// TIA Portal V21 export
FUNCTION_BLOCK "AiFb"   // FB108, LAD
{ S7_Optimized_Access := 'TRUE' }
// stored: AutoNumber false, MemoryReserve 100, SetENOAutomatically false
   VAR
      Ai01 { S7_SetPoint := 'True'} : "FB:Analog_Scaling";   // NfcoLineTemp(Ticr01)
      Ai02 { S7_SetPoint := 'True'} : "FB:Analog_Scaling";   // VfcoLineTemp(Ticr02)
      Ai03 { S7_SetPoint := 'True'} : "FB:Analog_Scaling";   // AiSpare01
      Ai04 { S7_SetPoint := 'True'} : "FB:Analog_Scaling";   // AiSpare02
      Ai05 { S7_SetPoint := 'True'} : "FB:Analog_Scaling";   // AiSpare03
      Ai06 { S7_SetPoint := 'True'} : "FB:Analog_Scaling";   // Pf01InLineTemp(Ticr06)
      Ai07 { S7_SetPoint := 'True'} : "FB:Analog_Scaling";   // Pf02InLineTemp(Ticr07)
      Ai08 { S7_SetPoint := 'True'} : "FB:Analog_Scaling";   // Pf02OutLineTemp(Ticr08)
      Ai09 { S7_SetPoint := 'True'} : "FB:Analog_Scaling";   // PtlDrainTemp(Ticr09)
      Ai10 { S7_SetPoint := 'True'} : "FB:Analog_Scaling";   // VesselTemp(Ticr10)
      Ai11 { S7_SetPoint := 'True'} : "FB:Analog_Scaling";   // VesselPressure(Picr01)
      Ai12 { S7_SetPoint := 'True'} : "FB:Analog_Scaling";   // VesselRclLine(Picr02)
      Ai13 { S7_SetPoint := 'True'} : "FB:Analog_Scaling";   // Pf01OutLinePressure(Picr03)
      Ai14 { S7_SetPoint := 'True'} : "FB:Analog_Scaling";   // Pf02OutLinePressure(Picr04)
      Ai15 { S7_SetPoint := 'True'} : "FB:Analog_Scaling";   // ProcessDrainConductivity
      Ai16 { S7_SetPoint := 'True'} : "FB:Analog_Scaling";   // AiSpare04
      Ai17 { S7_SetPoint := 'True'} : "FB:Analog_Scaling";   // AiSpare05
      Ai18 { S7_SetPoint := 'True'} : "FB:Analog_Scaling";   // AiSpare06
      Ai19 { S7_SetPoint := 'True'} : "FB:Analog_Scaling";   // AiSpare07
      Ai20 { S7_SetPoint := 'True'} : "FB:Analog_Scaling";   // AiSpare08
      Ai21 { S7_SetPoint := 'True'} : "FB:Analog_Scaling";   // AiSpare09
      Ai22 { S7_SetPoint := 'True'} : "FB:Analog_Scaling";   // AiSpare10
      Ai23 { S7_SetPoint := 'True'} : "FB:Analog_Scaling";   // AiSpare11
      Ai24 { S7_SetPoint := 'True'} : "FB:Analog_Scaling";   // AiSpare12
   END_VAR
BEGIN

REGION Network 1: #Ai01--- NfcoLineTemp
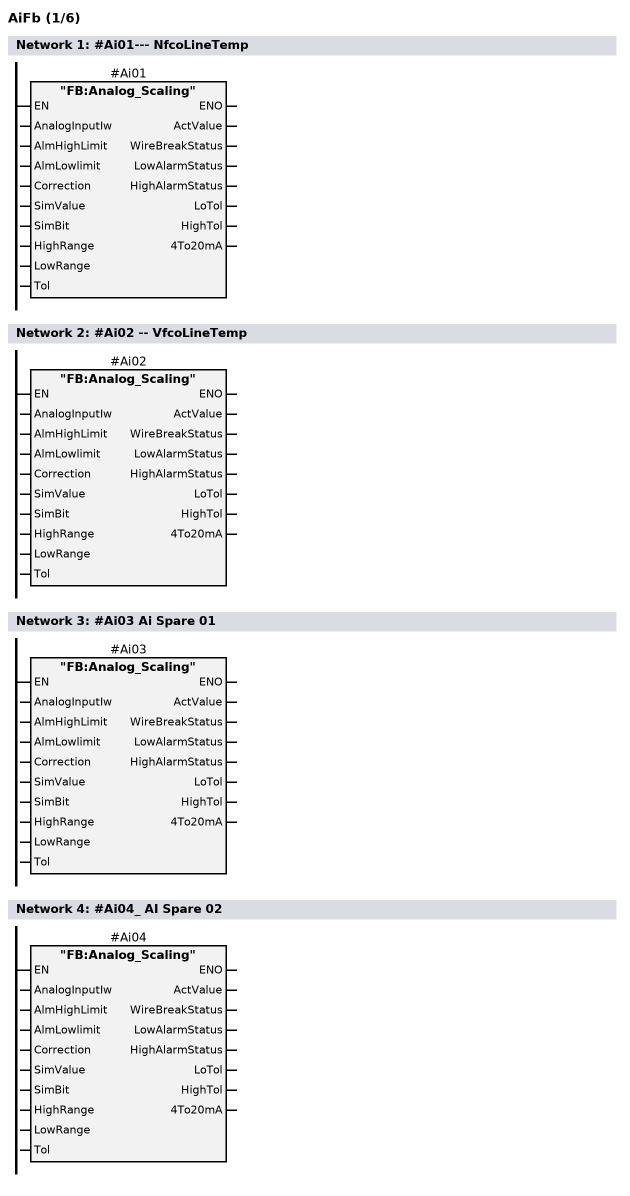
   RUNG wire#powerrail
      #Ai01(AnalogInputIw :=, AlmHighLimit :=, AlmLowlimit :=, Correction :=, SimValue :=, SimBit :=, HighRange :=, LowRange :=, Tol :=, ActValue =>, WireBreakStatus =>, LowAlarmStatus =>, HighAlarmStatus =>, LoTol =>, HighTol =>, "4To20mA" =>)
   END_RUNG
   // the same network as SCL:
   #Ai01();   // "FB:Analog_Scaling"
END_REGION

REGION Network 2: #Ai02 -- VfcoLineTemp
   RUNG wire#powerrail
      #Ai02(AnalogInputIw :=, AlmHighLimit :=, AlmLowlimit :=, Correction :=, SimValue :=, SimBit :=, HighRange :=, LowRange :=, Tol :=, ActValue =>, WireBreakStatus =>, LowAlarmStatus =>, HighAlarmStatus =>, LoTol =>, HighTol =>, "4To20mA" =>)
   END_RUNG
   // the same network as SCL:
   #Ai02();   // "FB:Analog_Scaling"
END_REGION

REGION Network 3: #Ai03 Ai Spare 01
   RUNG wire#powerrail
      #Ai03(AnalogInputIw :=, AlmHighLimit :=, AlmLowlimit :=, Correction :=, SimValue :=, SimBit :=, HighRange :=, LowRange :=, Tol :=, ActValue =>, WireBreakStatus =>, LowAlarmStatus =>, HighAlarmStatus =>, LoTol =>, HighTol =>, "4To20mA" =>)
   END_RUNG
   // the same network as SCL:
   #Ai03();   // "FB:Analog_Scaling"
END_REGION

REGION Network 4: #Ai04_ AI Spare 02
   RUNG wire#powerrail
      #Ai04(AnalogInputIw :=, AlmHighLimit :=, AlmLowlimit :=, Correction :=, SimValue :=, SimBit :=, HighRange :=, LowRange :=, Tol :=, ActValue =>, WireBreakStatus =>, LowAlarmStatus =>, HighAlarmStatus =>, LoTol =>, HighTol =>, "4To20mA" =>)
   END_RUNG
   // the same network as SCL:
   #Ai04();   // "FB:Analog_Scaling"
END_REGION

REGION Network 5: #Ai05--- #Ai04_ AI Spare 03
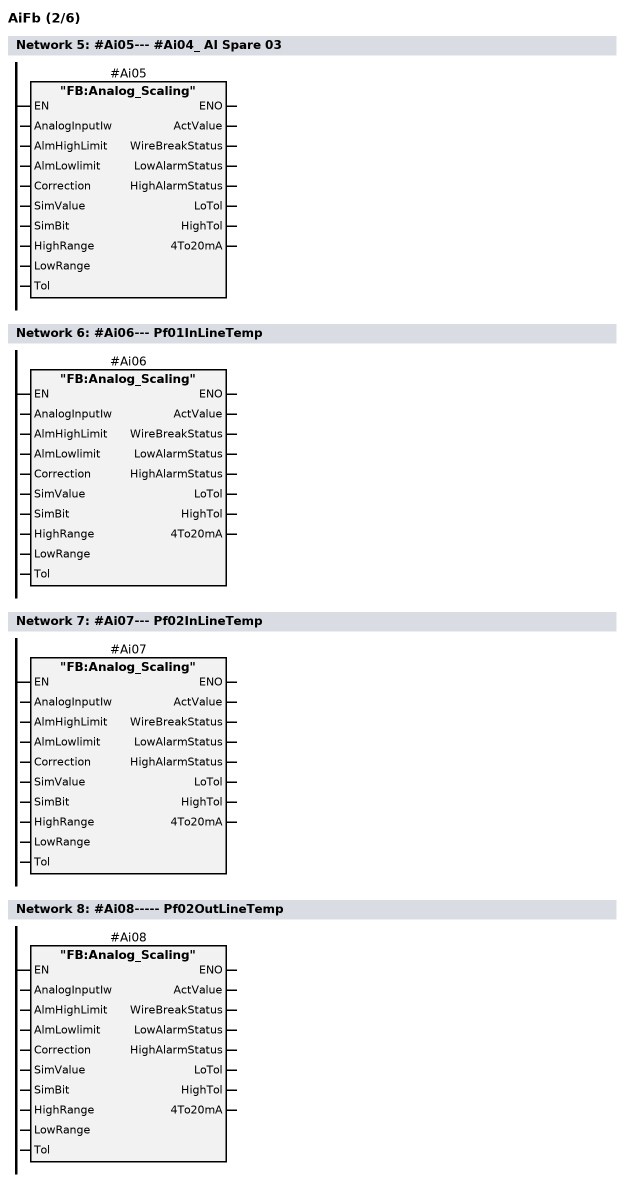
   RUNG wire#powerrail
      #Ai05(AnalogInputIw :=, AlmHighLimit :=, AlmLowlimit :=, Correction :=, SimValue :=, SimBit :=, HighRange :=, LowRange :=, Tol :=, ActValue =>, WireBreakStatus =>, LowAlarmStatus =>, HighAlarmStatus =>, LoTol =>, HighTol =>, "4To20mA" =>)
   END_RUNG
   // the same network as SCL:
   #Ai05();   // "FB:Analog_Scaling"
END_REGION

REGION Network 6: #Ai06--- Pf01InLineTemp
   RUNG wire#powerrail
      #Ai06(AnalogInputIw :=, AlmHighLimit :=, AlmLowlimit :=, Correction :=, SimValue :=, SimBit :=, HighRange :=, LowRange :=, Tol :=, ActValue =>, WireBreakStatus =>, LowAlarmStatus =>, HighAlarmStatus =>, LoTol =>, HighTol =>, "4To20mA" =>)
   END_RUNG
   // the same network as SCL:
   #Ai06();   // "FB:Analog_Scaling"
END_REGION

REGION Network 7: #Ai07--- Pf02InLineTemp
   RUNG wire#powerrail
      #Ai07(AnalogInputIw :=, AlmHighLimit :=, AlmLowlimit :=, Correction :=, SimValue :=, SimBit :=, HighRange :=, LowRange :=, Tol :=, ActValue =>, WireBreakStatus =>, LowAlarmStatus =>, HighAlarmStatus =>, LoTol =>, HighTol =>, "4To20mA" =>)
   END_RUNG
   // the same network as SCL:
   #Ai07();   // "FB:Analog_Scaling"
END_REGION

REGION Network 8: #Ai08----- Pf02OutLineTemp
   RUNG wire#powerrail
      #Ai08(AnalogInputIw :=, AlmHighLimit :=, AlmLowlimit :=, Correction :=, SimValue :=, SimBit :=, HighRange :=, LowRange :=, Tol :=, ActValue =>, WireBreakStatus =>, LowAlarmStatus =>, HighAlarmStatus =>, LoTol =>, HighTol =>, "4To20mA" =>)
   END_RUNG
   // the same network as SCL:
   #Ai08();   // "FB:Analog_Scaling"
END_REGION

REGION Network 9: #Ai09---- PtlDrainTemp
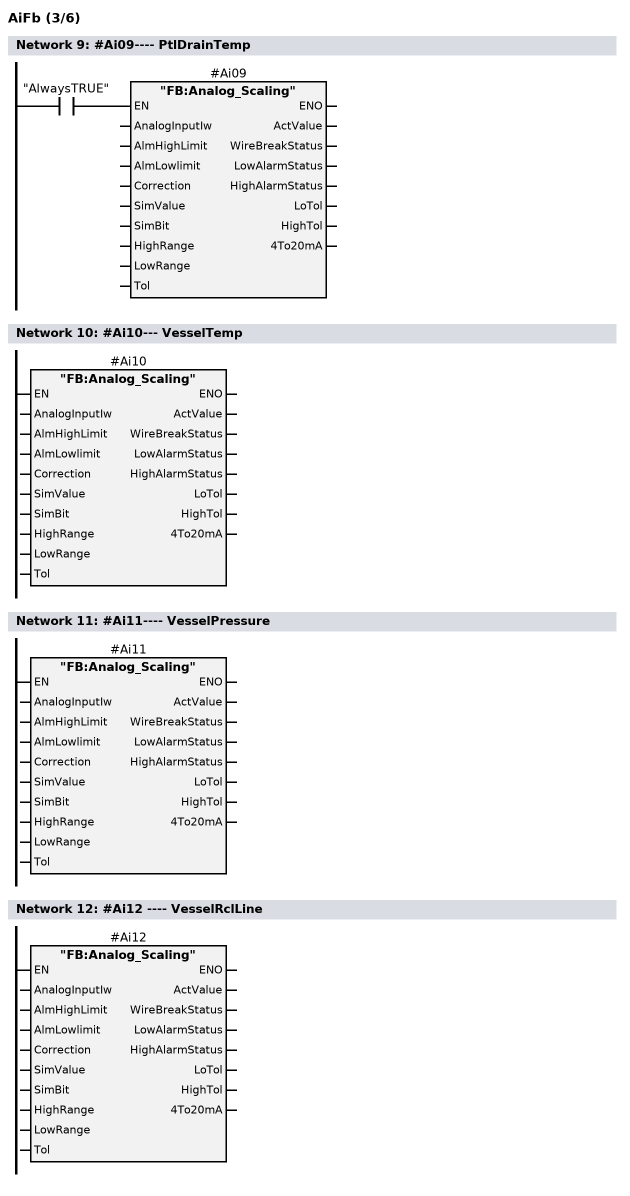
   RUNG wire#powerrail
      Contact( "AlwaysTRUE" )
      #Ai09(AnalogInputIw :=, AlmHighLimit :=, AlmLowlimit :=, Correction :=, SimValue :=, SimBit :=, HighRange :=, LowRange :=, Tol :=, ActValue =>, WireBreakStatus =>, LowAlarmStatus =>, HighAlarmStatus =>, LoTol =>, HighTol =>, "4To20mA" =>)
   END_RUNG
   // the same network as SCL:
   IF "AlwaysTRUE" THEN
       #Ai09();   // "FB:Analog_Scaling"
   END_IF;
END_REGION

REGION Network 10: #Ai10--- VesselTemp
   RUNG wire#powerrail
      #Ai10(AnalogInputIw :=, AlmHighLimit :=, AlmLowlimit :=, Correction :=, SimValue :=, SimBit :=, HighRange :=, LowRange :=, Tol :=, ActValue =>, WireBreakStatus =>, LowAlarmStatus =>, HighAlarmStatus =>, LoTol =>, HighTol =>, "4To20mA" =>)
   END_RUNG
   // the same network as SCL:
   #Ai10();   // "FB:Analog_Scaling"
END_REGION

REGION Network 11: #Ai11---- VesselPressure
   RUNG wire#powerrail
      #Ai11(AnalogInputIw :=, AlmHighLimit :=, AlmLowlimit :=, Correction :=, SimValue :=, SimBit :=, HighRange :=, LowRange :=, Tol :=, ActValue =>, WireBreakStatus =>, LowAlarmStatus =>, HighAlarmStatus =>, LoTol =>, HighTol =>, "4To20mA" =>)
   END_RUNG
   // the same network as SCL:
   #Ai11();   // "FB:Analog_Scaling"
END_REGION

REGION Network 12: #Ai12 ---- VesselRclLine
   RUNG wire#powerrail
      #Ai12(AnalogInputIw :=, AlmHighLimit :=, AlmLowlimit :=, Correction :=, SimValue :=, SimBit :=, HighRange :=, LowRange :=, Tol :=, ActValue =>, WireBreakStatus =>, LowAlarmStatus =>, HighAlarmStatus =>, LoTol =>, HighTol =>, "4To20mA" =>)
   END_RUNG
   // the same network as SCL:
   #Ai12();   // "FB:Analog_Scaling"
END_REGION

REGION Network 13: #Ai13--- Pf01OutLinePressure
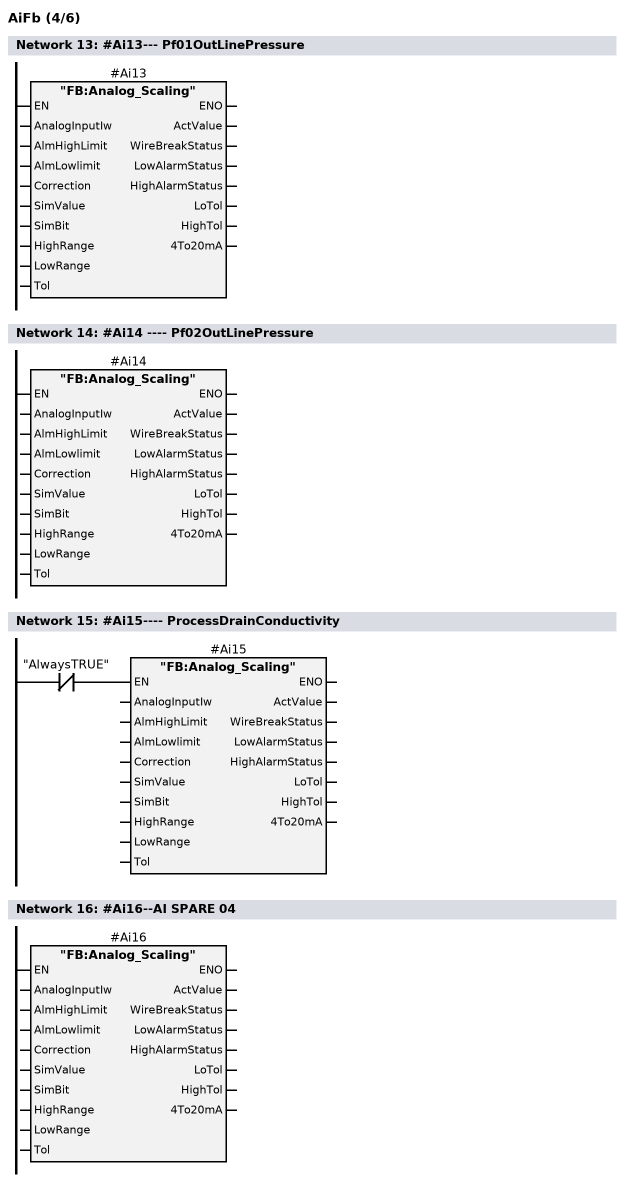
   RUNG wire#powerrail
      #Ai13(AnalogInputIw :=, AlmHighLimit :=, AlmLowlimit :=, Correction :=, SimValue :=, SimBit :=, HighRange :=, LowRange :=, Tol :=, ActValue =>, WireBreakStatus =>, LowAlarmStatus =>, HighAlarmStatus =>, LoTol =>, HighTol =>, "4To20mA" =>)
   END_RUNG
   // the same network as SCL:
   #Ai13();   // "FB:Analog_Scaling"
END_REGION

REGION Network 14: #Ai14 ---- Pf02OutLinePressure
   RUNG wire#powerrail
      #Ai14(AnalogInputIw :=, AlmHighLimit :=, AlmLowlimit :=, Correction :=, SimValue :=, SimBit :=, HighRange :=, LowRange :=, Tol :=, ActValue =>, WireBreakStatus =>, LowAlarmStatus =>, HighAlarmStatus =>, LoTol =>, HighTol =>, "4To20mA" =>)
   END_RUNG
   // the same network as SCL:
   #Ai14();   // "FB:Analog_Scaling"
END_REGION

REGION Network 15: #Ai15---- ProcessDrainConductivity
   RUNG wire#powerrail
      I_Contact( "AlwaysTRUE" )
      #Ai15(AnalogInputIw :=, AlmHighLimit :=, AlmLowlimit :=, Correction :=, SimValue :=, SimBit :=, HighRange :=, LowRange :=, Tol :=, ActValue =>, WireBreakStatus =>, LowAlarmStatus =>, HighAlarmStatus =>, LoTol =>, HighTol =>, "4To20mA" =>)
   END_RUNG
   // the same network as SCL:
   IF NOT "AlwaysTRUE" THEN
       #Ai15();   // "FB:Analog_Scaling"
   END_IF;
END_REGION

REGION Network 16: #Ai16--AI SPARE 04
   RUNG wire#powerrail
      #Ai16(AnalogInputIw :=, AlmHighLimit :=, AlmLowlimit :=, Correction :=, SimValue :=, SimBit :=, HighRange :=, LowRange :=, Tol :=, ActValue =>, WireBreakStatus =>, LowAlarmStatus =>, HighAlarmStatus =>, LoTol =>, HighTol =>, "4To20mA" =>)
   END_RUNG
   // the same network as SCL:
   #Ai16();   // "FB:Analog_Scaling"
END_REGION

REGION Network 17: #Ai17--AI SPARE 05
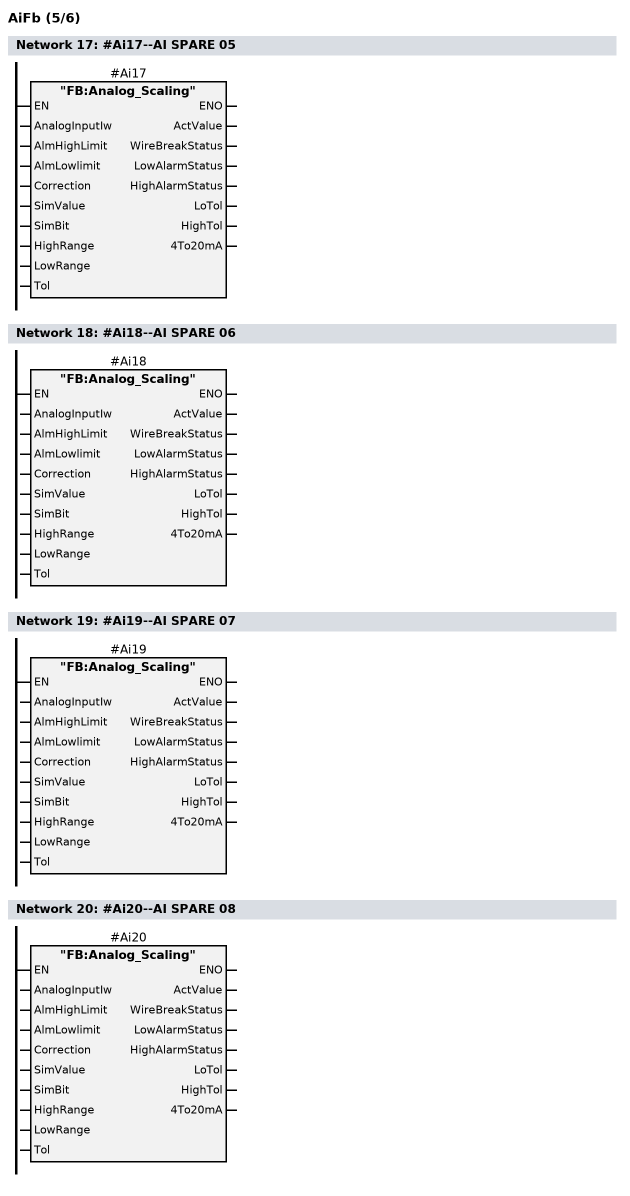
   RUNG wire#powerrail
      #Ai17(AnalogInputIw :=, AlmHighLimit :=, AlmLowlimit :=, Correction :=, SimValue :=, SimBit :=, HighRange :=, LowRange :=, Tol :=, ActValue =>, WireBreakStatus =>, LowAlarmStatus =>, HighAlarmStatus =>, LoTol =>, HighTol =>, "4To20mA" =>)
   END_RUNG
   // the same network as SCL:
   #Ai17();   // "FB:Analog_Scaling"
END_REGION

REGION Network 18: #Ai18--AI SPARE 06
   RUNG wire#powerrail
      #Ai18(AnalogInputIw :=, AlmHighLimit :=, AlmLowlimit :=, Correction :=, SimValue :=, SimBit :=, HighRange :=, LowRange :=, Tol :=, ActValue =>, WireBreakStatus =>, LowAlarmStatus =>, HighAlarmStatus =>, LoTol =>, HighTol =>, "4To20mA" =>)
   END_RUNG
   // the same network as SCL:
   #Ai18();   // "FB:Analog_Scaling"
END_REGION

REGION Network 19: #Ai19--AI SPARE 07
   RUNG wire#powerrail
      #Ai19(AnalogInputIw :=, AlmHighLimit :=, AlmLowlimit :=, Correction :=, SimValue :=, SimBit :=, HighRange :=, LowRange :=, Tol :=, ActValue =>, WireBreakStatus =>, LowAlarmStatus =>, HighAlarmStatus =>, LoTol =>, HighTol =>, "4To20mA" =>)
   END_RUNG
   // the same network as SCL:
   #Ai19();   // "FB:Analog_Scaling"
END_REGION

REGION Network 20: #Ai20--AI SPARE 08
   RUNG wire#powerrail
      #Ai20(AnalogInputIw :=, AlmHighLimit :=, AlmLowlimit :=, Correction :=, SimValue :=, SimBit :=, HighRange :=, LowRange :=, Tol :=, ActValue =>, WireBreakStatus =>, LowAlarmStatus =>, HighAlarmStatus =>, LoTol =>, HighTol =>, "4To20mA" =>)
   END_RUNG
   // the same network as SCL:
   #Ai20();   // "FB:Analog_Scaling"
END_REGION

REGION Network 21: #Ai21--AI SPARE 09
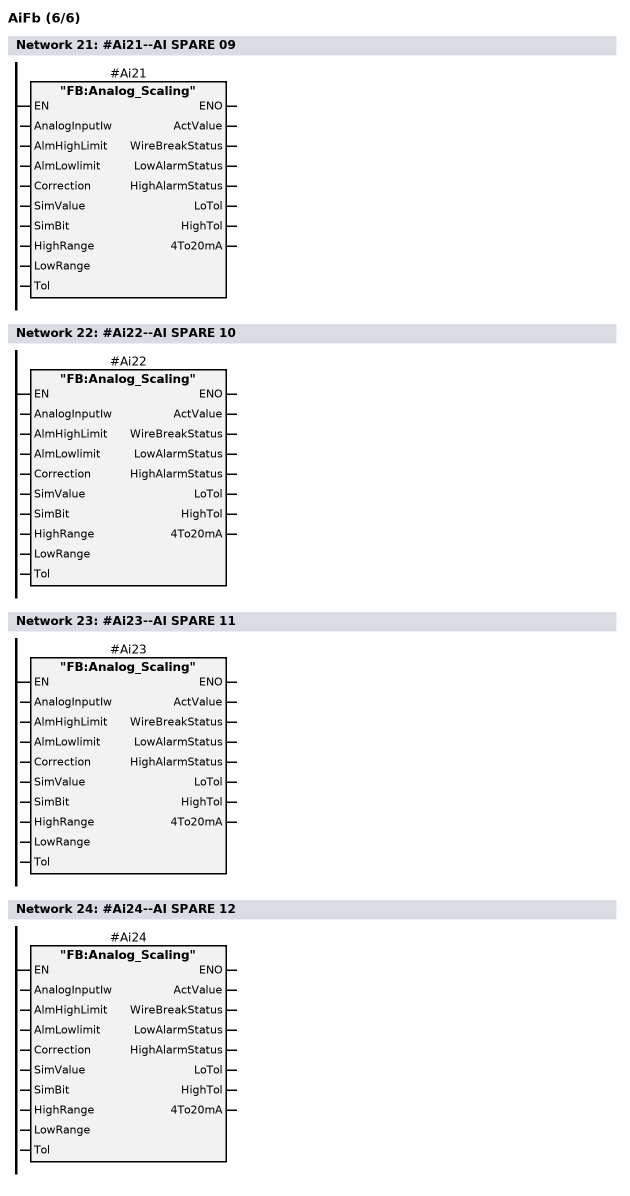
   RUNG wire#powerrail
      #Ai21(AnalogInputIw :=, AlmHighLimit :=, AlmLowlimit :=, Correction :=, SimValue :=, SimBit :=, HighRange :=, LowRange :=, Tol :=, ActValue =>, WireBreakStatus =>, LowAlarmStatus =>, HighAlarmStatus =>, LoTol =>, HighTol =>, "4To20mA" =>)
   END_RUNG
   // the same network as SCL:
   #Ai21();   // "FB:Analog_Scaling"
END_REGION

REGION Network 22: #Ai22--AI SPARE 10
   RUNG wire#powerrail
      #Ai22(AnalogInputIw :=, AlmHighLimit :=, AlmLowlimit :=, Correction :=, SimValue :=, SimBit :=, HighRange :=, LowRange :=, Tol :=, ActValue =>, WireBreakStatus =>, LowAlarmStatus =>, HighAlarmStatus =>, LoTol =>, HighTol =>, "4To20mA" =>)
   END_RUNG
   // the same network as SCL:
   #Ai22();   // "FB:Analog_Scaling"
END_REGION

REGION Network 23: #Ai23--AI SPARE 11
   RUNG wire#powerrail
      #Ai23(AnalogInputIw :=, AlmHighLimit :=, AlmLowlimit :=, Correction :=, SimValue :=, SimBit :=, HighRange :=, LowRange :=, Tol :=, ActValue =>, WireBreakStatus =>, LowAlarmStatus =>, HighAlarmStatus =>, LoTol =>, HighTol =>, "4To20mA" =>)
   END_RUNG
   // the same network as SCL:
   #Ai23();   // "FB:Analog_Scaling"
END_REGION

REGION Network 24: #Ai24--AI SPARE 12
   RUNG wire#powerrail
      #Ai24(AnalogInputIw :=, AlmHighLimit :=, AlmLowlimit :=, Correction :=, SimValue :=, SimBit :=, HighRange :=, LowRange :=, Tol :=, ActValue =>, WireBreakStatus =>, LowAlarmStatus =>, HighAlarmStatus =>, LoTol =>, HighTol =>, "4To20mA" =>)
   END_RUNG
   // the same network as SCL:
   #Ai24();   // "FB:Analog_Scaling"
END_REGION
END_FUNCTION_BLOCK
